INTERFACE itfDetect

PROPERTY pDetectSignal : BOOL
GET
END_GET
SET
END_SET
END_PROPERTY

END_INTERFACE

(* stored: Version 1.1.0.1, ProductVersion 3.1.4024.12
   Itf itfDetect: Id {708b1dff-bdc8-4e79-bc34-4b561f8c1fcb}
   Property pDetectSignal: Id {49f8113c-e4d4-4f1b-8a62-312c2136cc10}
   Get Get: Id {9a8a69e0-a62c-48ac-87dc-71ffead1bd87}
   Set Set: Id {e67219b9-137c-4820-93f0-b3c172fb3f50} *)
